{attribute 'GeneratedUsingTerminal: KL8001'}
{attribute addProperty BoxType "KL8001"}
{attribute addProperty Id "Channel_1AT %Q*Channel_D9D488070"}
{attribute addProperty CRC "2002871610"}
{attribute addProperty Size "0"}
TYPE KL8001_7761653A :
STRUCT
	{attribute addProperty Name "Channel_1"}
	Channel_1 : Channel_D9D48807;
END_STRUCT
END_TYPE

(* stored: Version 1.2.0.0, ProductVersion 3.1.4024.9
   DUT KL8001_7761653A: Id {5ef6c84d-c347-4ebf-9238-a569c7277700} *)
